Staubli VAL3: TxtReadRoom1.pgx

program TxtReadRoom1()
  local string l_str
  local num nNumpoint
  local num ntext
  local string sTxtfile
begin
  bTxt1=false
  delay(0)
  l_str=toString("1",n_sTxt)
  sTxtfile="path"+l_str+".txt"
  ntext=$fileOpen(sTxtfile,"r")
  for nNumpoint=0 to 499
    $fileGet(ntext,sString[nNumpoint],1)
    if sString[nNumpoint]!=""
      call stringtopoint(sString[nNumpoint],nNumpoint)
    else
    endIf
  endFor
  delay(0)


  if n_sTxt==nTxtTotal-1
    n_sTxt=0
  elseIf n_sTxt!=nTxtTotal-1
    n_sTxt=n_sTxt+1
  endIf

  nNumpoint=nNumpoint-1
  $fileClose(ntext)
end
